GLOBALCONSTANTS ButtonActivationCode (* ButtonActivationCode constants *)
  (* Standard: 61499-1; Description: Copyright (c) 2024 HR Agrartechnik GmbH This program and the accompanying materials are made available under the terms of the Eclipse Public License 2.0 which is available at https://www.eclipse.org/legal/epl-2.0/ SPDX-License-Identifier: EPL-2.0 *)
  (* Version 1.0, 2024-01-25, Franz Höpfinger, HR Agrartechnik GmbH *)
  PACKAGE isobus::UT::io::Button;
  VAR_GLOBAL CONSTANT
    BT_RELEASED_UNLATCHED : isobus::UT::io::Button::ButtonActivationCode_S := (code := 0); (* Button has been unlatched or released (state change) *)
    BT_PRESSED_LATCHED : isobus::UT::io::Button::ButtonActivationCode_S := (code := 1); (* Button has been “pressed” or latched (state change) *)
    BT_STILL_HELD : isobus::UT::io::Button::ButtonActivationCode_S := (code := 2); (* Button is still held (latchable buttons do not repeat) *)
    BT_STILL_HELD_START : isobus::UT::io::Button::ButtonActivationCode_S := (code := 2, bCyclic := FALSE); (* Button is still held (latchable buttons do not repeat) *)
    BT_ABORTED : isobus::UT::io::Button::ButtonActivationCode_S := (code := 3); (* Button press aborted (Applies to VT version 4 and later) *)
    Invalid : isobus::UT::io::Button::ButtonActivationCode_S := (code := 255);
  END_VAR
END_GLOBALCONSTANTS
